SYSTEM ETFA2023
  (* Version 1.0, 2023-03-17, AK125171 *)
  APPLICATION ETFA2023App
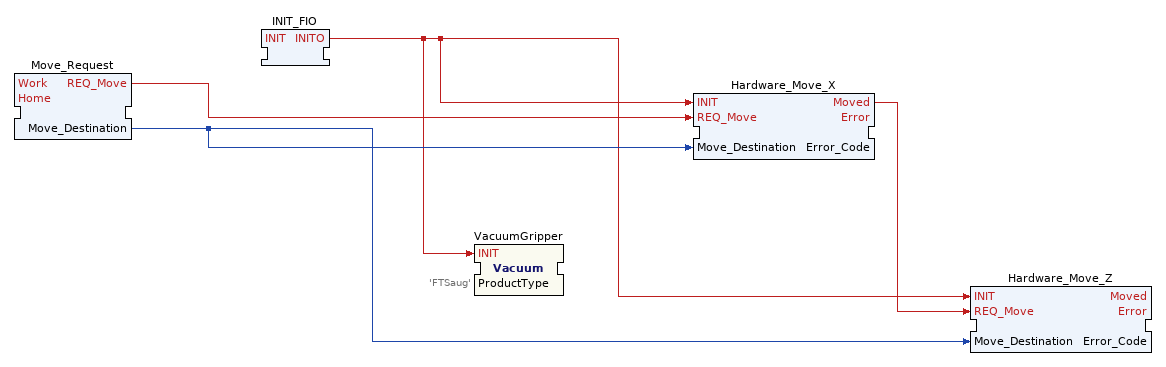
    FBS
      VacuumGripper : Vacuum(ProductType := 'FTSaug');
    END_FBS
    SUBAPPLICATION INIT_FIO
      EVENT_INPUT
        INIT;
      END_EVENT
      EVENT_OUTPUT
        INITO;
      END_EVENT
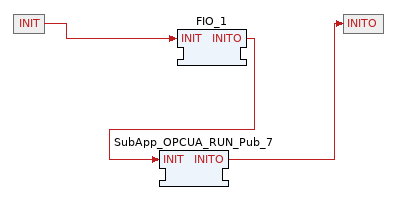
      SUBAPPLICATION SubApp_OPCUA_RUN_Pub_7
        EVENT_INPUT
          INIT;
        END_EVENT
        EVENT_OUTPUT
          INITO;
        END_EVENT
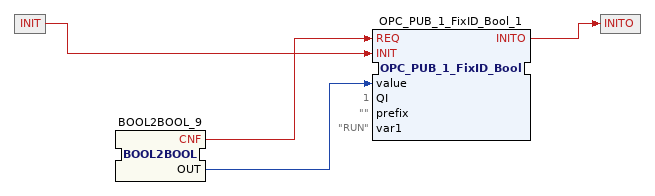
        FBS
          BOOL2BOOL_9 : BOOL2BOOL;
        END_FBS
        SUBAPPS
          OPC_PUB_1_FixID_Bool_1 : OPC_PUB_1_FixID_Bool(QI := 1, prefix := "", var1 := "RUN");
        END_SUBAPPS
        EVENT_CONNECTIONS
          BOOL2BOOL_9.CNF TO OPC_PUB_1_FixID_Bool_1.REQ;
          INIT TO OPC_PUB_1_FixID_Bool_1.INIT;
          OPC_PUB_1_FixID_Bool_1.INITO TO INITO;
        END_CONNECTIONS
        DATA_CONNECTIONS
          BOOL2BOOL_9.OUT TO OPC_PUB_1_FixID_Bool_1.value;
        END_CONNECTIONS
      END_SUBAPPLICATION
      SUBAPPLICATION FIO_1
        EVENT_INPUT
          INIT;
        END_EVENT
        EVENT_OUTPUT
          INITO;
        END_EVENT
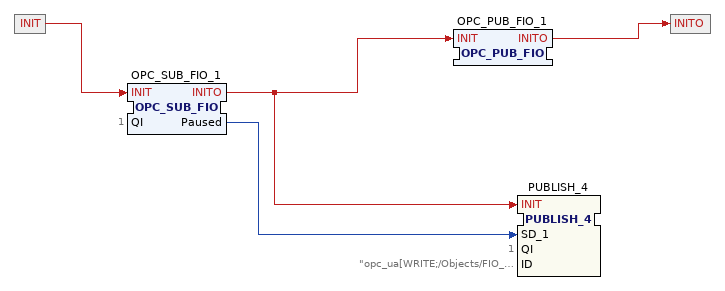
        FBS
          PUBLISH_4 : PUBLISH_4(QI := 1, ID := "opc_ua[WRITE;/Objects/FIO_Q_CameraPosition, 1:s=FIO_Q_CameraPosition;/Objects/FIO_Q_Pause, 1:s=FIO_Q_Pause;/Objects/FIO_Q_Reset, 1:s=FIO_Q_Reset;/Objects/FIO_Q_Run, 1:s=FIO_Q_Run]");
        END_FBS
        SUBAPPS
          OPC_PUB_FIO_1 : OPC_PUB_FIO;
          OPC_SUB_FIO_1 : OPC_SUB_FIO(QI := 1);
        END_SUBAPPS
        EVENT_CONNECTIONS
          OPC_SUB_FIO_1.INITO TO PUBLISH_4.INIT;
          OPC_SUB_FIO_1.INITO TO OPC_PUB_FIO_1.INIT;
          OPC_PUB_FIO_1.INITO TO INITO;
          INIT TO OPC_SUB_FIO_1.INIT;
        END_CONNECTIONS
        DATA_CONNECTIONS
          OPC_SUB_FIO_1.Paused TO PUBLISH_4.SD_1;
        END_CONNECTIONS
      END_SUBAPPLICATION
      EVENT_CONNECTIONS
        FIO_1.INITO TO SubApp_OPCUA_RUN_Pub_7.INIT;
        INIT TO FIO_1.INIT;
        SubApp_OPCUA_RUN_Pub_7.INITO TO INITO;
      END_CONNECTIONS
    END_SUBAPPLICATION
    SUBAPPLICATION Move_Request
      EVENT_INPUT
        Work;
        Home;
      END_EVENT
      EVENT_OUTPUT
        REQ_Move;
      END_EVENT
      VAR_OUTPUT
        Move_Destination : STRING;
      END_VAR
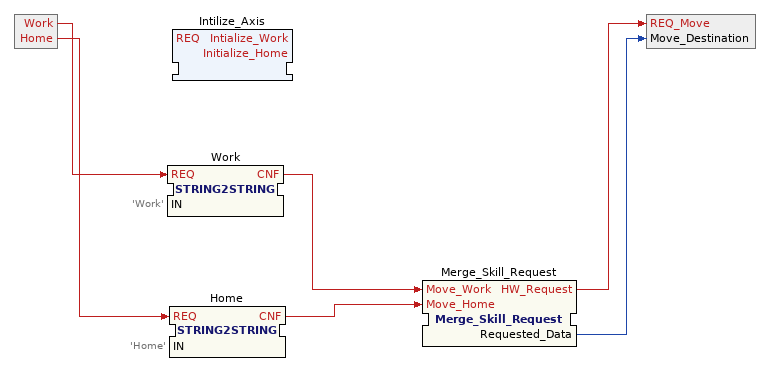
      FBS
        Work : STRING2STRING(IN := 'Work');
        Home : STRING2STRING(IN := 'Home');
        Merge_Skill_Request : Merge_Skill_Request;
      END_FBS
      SUBAPPLICATION Intilize_Axis
        EVENT_INPUT
          REQ;
        END_EVENT
        EVENT_OUTPUT
          Intialize_Work; (* Connect to Move_Work to intialize Work as start position else Connect to Move_Home to intialize Home as start position *)
          Initialize_Home;
        END_EVENT
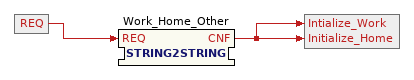
        FBS
          Work_Home_Other : STRING2STRING; (* Connect to Move_Work or Move_Home interface  of Instace Merge_Skill_Request *)
        END_FBS
        EVENT_CONNECTIONS
          REQ TO Work_Home_Other.REQ;
          Work_Home_Other.CNF TO Intialize_Work;
          Work_Home_Other.CNF TO Initialize_Home;
        END_CONNECTIONS
      END_SUBAPPLICATION
      EVENT_CONNECTIONS
        Work TO Work.REQ;
        Home TO Home.REQ;
        Work.CNF TO Merge_Skill_Request.Move_Work;
        Home.CNF TO Merge_Skill_Request.Move_Home;
        Merge_Skill_Request.HW_Request TO REQ_Move;
      END_CONNECTIONS
      DATA_CONNECTIONS
        Merge_Skill_Request.Requested_Data TO Move_Destination;
      END_CONNECTIONS
    END_SUBAPPLICATION
    SUBAPPLICATION Hardware_Move_X (* Hardware *)
      EVENT_INPUT
        INIT;
        REQ_Move;
      END_EVENT
      EVENT_OUTPUT
        Moved;
        Error;
      END_EVENT
      VAR_INPUT
        Move_Destination : STRING;
      END_VAR
      VAR_OUTPUT
        Error_Code : INT;
      END_VAR
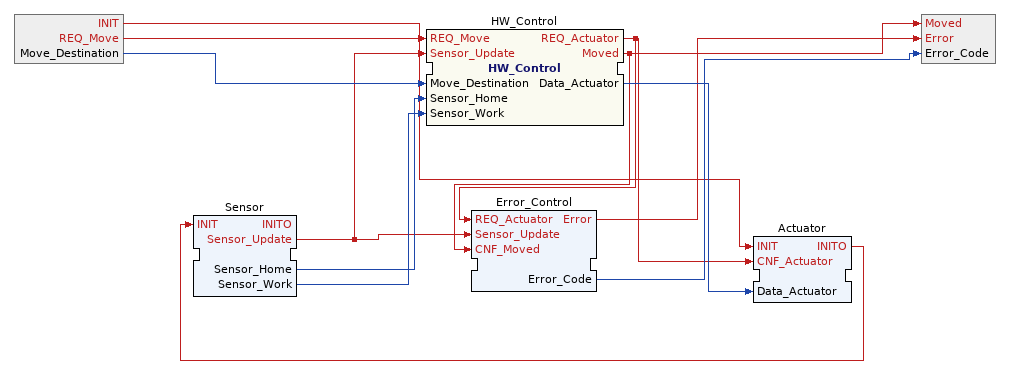
      FBS
        HW_Control : HW_Control;
      END_FBS
      SUBAPPLICATION Actuator
        EVENT_INPUT
          INIT;
          CNF_Actuator;
        END_EVENT
        EVENT_OUTPUT
          INITO;
        END_EVENT
        VAR_INPUT
          Data_Actuator : BOOL;
        END_VAR
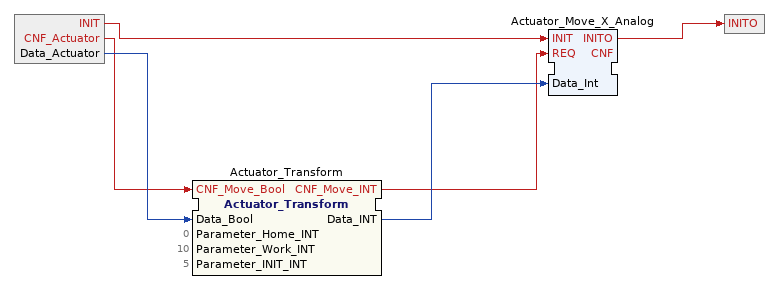
        FBS
          Actuator_Transform : Actuator_Transform(Parameter_Home_INT := 0, Parameter_Work_INT := 10, Parameter_INIT_INT := 5);
        END_FBS
        SUBAPPLICATION Actuator_Move_X_Analog
          EVENT_INPUT
            INIT;
            REQ;
          END_EVENT
          EVENT_OUTPUT
            INITO;
            CNF;
          END_EVENT
          VAR_INPUT
            Data_Int : INT;
          END_VAR
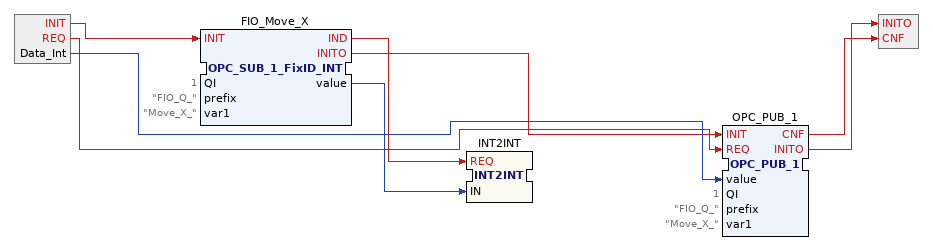
          FBS
            INT2INT : INT2INT;
          END_FBS
          SUBAPPS
            FIO_Move_X : OPC_SUB_1_FixID_INT(QI := 1, prefix := "FIO_Q_", var1 := "Move_X_");
            OPC_PUB_1 : OPC_PUB_1(QI := 1, prefix := "FIO_Q_", var1 := "Move_X_");
          END_SUBAPPS
          EVENT_CONNECTIONS
            INIT TO FIO_Move_X.INIT;
            FIO_Move_X.IND TO INT2INT.REQ;
            FIO_Move_X.INITO TO OPC_PUB_1.INIT;
            OPC_PUB_1.CNF TO CNF;
            OPC_PUB_1.INITO TO INITO;
            REQ TO OPC_PUB_1.REQ;
          END_CONNECTIONS
          DATA_CONNECTIONS
            Data_Int TO OPC_PUB_1.value;
            FIO_Move_X.value TO INT2INT.IN;
          END_CONNECTIONS
        END_SUBAPPLICATION
        EVENT_CONNECTIONS
          INIT TO Actuator_Move_X_Analog.INIT;
          Actuator_Move_X_Analog.INITO TO INITO;
          CNF_Actuator TO Actuator_Transform.CNF_Move_Bool;
          Actuator_Transform.CNF_Move_INT TO Actuator_Move_X_Analog.REQ;
        END_CONNECTIONS
        DATA_CONNECTIONS
          Data_Actuator TO Actuator_Transform.Data_Bool;
          Actuator_Transform.Data_INT TO Actuator_Move_X_Analog.Data_Int;
        END_CONNECTIONS
      END_SUBAPPLICATION
      SUBAPPLICATION Error_Control
        EVENT_INPUT
          REQ_Actuator;
          Sensor_Update;
          CNF_Moved;
        END_EVENT
        EVENT_OUTPUT
          Error;
        END_EVENT
        VAR_OUTPUT
          Error_Code : INT; (* Error_Code_1_For_Movement_Not_Started_Error_Code_2_For_Movement_Timing *)
        END_VAR
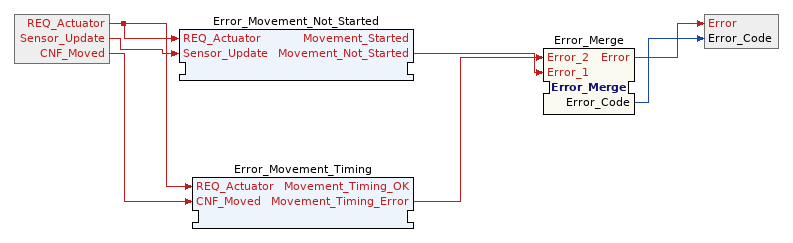
        FBS
          Error_Merge : Error_Merge;
        END_FBS
        SUBAPPLICATION Error_Movement_Not_Started
          EVENT_INPUT
            REQ_Actuator;
            Sensor_Update;
          END_EVENT
          EVENT_OUTPUT
            Movement_Started;
            Movement_Not_Started;
          END_EVENT
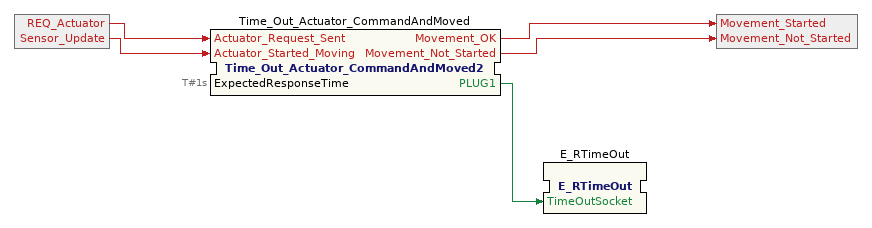
          FBS
            E_RTimeOut : E_RTimeOut;
            Time_Out_Actuator_CommandAndMoved : Time_Out_Actuator_CommandAndMoved2(ExpectedResponseTime := T#1s);
          END_FBS
          EVENT_CONNECTIONS
            REQ_Actuator TO Time_Out_Actuator_CommandAndMoved.Actuator_Request_Sent;
            Sensor_Update TO Time_Out_Actuator_CommandAndMoved.Actuator_Started_Moving;
            Time_Out_Actuator_CommandAndMoved.Movement_OK TO Movement_Started;
            Time_Out_Actuator_CommandAndMoved.Movement_Not_Started TO Movement_Not_Started;
          END_CONNECTIONS
          ADAPTER_CONNECTIONS
            Time_Out_Actuator_CommandAndMoved.PLUG1 TO E_RTimeOut.TimeOutSocket;
          END_CONNECTIONS
        END_SUBAPPLICATION
        SUBAPPLICATION Error_Movement_Timing
          EVENT_INPUT
            REQ_Actuator;
            CNF_Moved;
          END_EVENT
          EVENT_OUTPUT
            Movement_Timing_OK;
            Movement_Timing_Error;
          END_EVENT
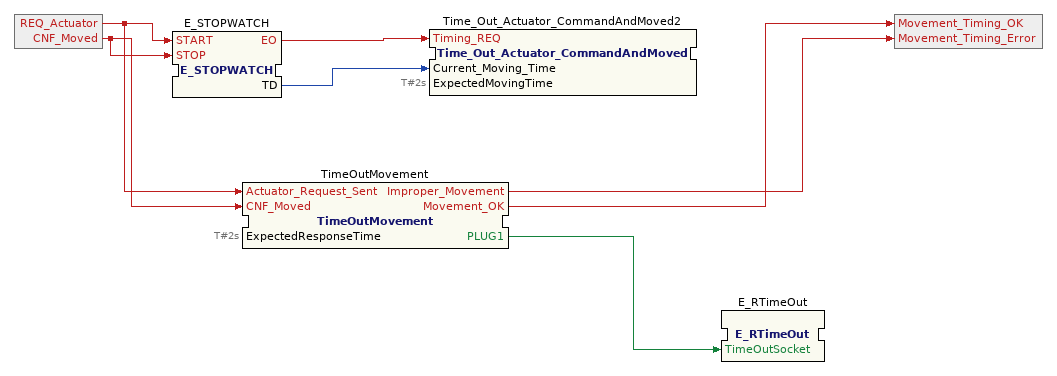
          FBS
            E_STOPWATCH : E_STOPWATCH;
            Time_Out_Actuator_CommandAndMoved2 : Time_Out_Actuator_CommandAndMoved(ExpectedMovingTime := T#2s);
            E_RTimeOut : E_RTimeOut;
            TimeOutMovement : TimeOutMovement(ExpectedResponseTime := T#2s);
          END_FBS
          EVENT_CONNECTIONS
            E_STOPWATCH.EO TO Time_Out_Actuator_CommandAndMoved2.Timing_REQ;
            REQ_Actuator TO TimeOutMovement.Actuator_Request_Sent;
            CNF_Moved TO TimeOutMovement.CNF_Moved;
            TimeOutMovement.Improper_Movement TO Movement_Timing_Error;
            TimeOutMovement.Movement_OK TO Movement_Timing_OK;
            REQ_Actuator TO E_STOPWATCH.START;
            CNF_Moved TO E_STOPWATCH.STOP;
          END_CONNECTIONS
          DATA_CONNECTIONS
            E_STOPWATCH.TD TO Time_Out_Actuator_CommandAndMoved2.Current_Moving_Time;
          END_CONNECTIONS
          ADAPTER_CONNECTIONS
            TimeOutMovement.PLUG1 TO E_RTimeOut.TimeOutSocket;
          END_CONNECTIONS
        END_SUBAPPLICATION
        EVENT_CONNECTIONS
          REQ_Actuator TO Error_Movement_Not_Started.REQ_Actuator;
          Sensor_Update TO Error_Movement_Not_Started.Sensor_Update;
          CNF_Moved TO Error_Movement_Timing.CNF_Moved;
          Error_Movement_Timing.Movement_Timing_Error TO Error_Merge.Error_2;
          Error_Merge.Error TO Error;
          Error_Movement_Not_Started.Movement_Not_Started TO Error_Merge.Error_1;
          REQ_Actuator TO Error_Movement_Timing.REQ_Actuator;
        END_CONNECTIONS
        DATA_CONNECTIONS
          Error_Merge.Error_Code TO Error_Code;
        END_CONNECTIONS
      END_SUBAPPLICATION
      SUBAPPLICATION Sensor
        EVENT_INPUT
          INIT;
        END_EVENT
        EVENT_OUTPUT
          INITO;
          Sensor_Update;
        END_EVENT
        VAR_OUTPUT
          Sensor_Home : BOOL;
          Sensor_Work : BOOL;
        END_VAR
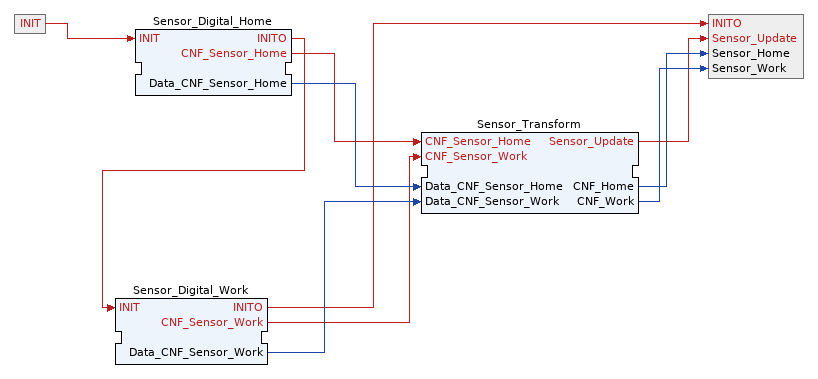
        SUBAPPLICATION Sensor_Digital_Work
          EVENT_INPUT
            INIT;
          END_EVENT
          EVENT_OUTPUT
            INITO;
            CNF_Sensor_Work;
          END_EVENT
          VAR_OUTPUT
            Data_CNF_Sensor_Work : BOOL;
          END_VAR
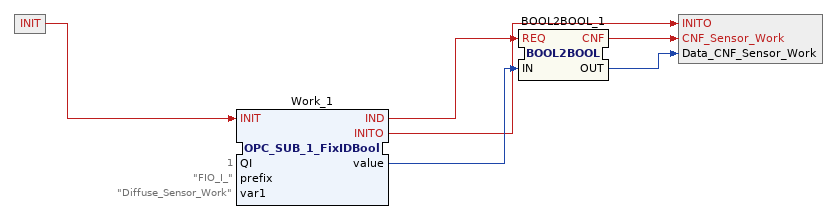
          FBS
            BOOL2BOOL_1 : BOOL2BOOL;
          END_FBS
          SUBAPPS
            Work_1 : OPC_SUB_1_FixIDBool(QI := 1, prefix := "FIO_I_", var1 := "Diffuse_Sensor_Work");
          END_SUBAPPS
          EVENT_CONNECTIONS
            Work_1.IND TO BOOL2BOOL_1.REQ;
            INIT TO Work_1.INIT;
            Work_1.INITO TO INITO;
            BOOL2BOOL_1.CNF TO CNF_Sensor_Work;
          END_CONNECTIONS
          DATA_CONNECTIONS
            Work_1.value TO BOOL2BOOL_1.IN;
            BOOL2BOOL_1.OUT TO Data_CNF_Sensor_Work;
          END_CONNECTIONS
        END_SUBAPPLICATION
        SUBAPPLICATION Sensor_Digital_Home
          EVENT_INPUT
            INIT;
          END_EVENT
          EVENT_OUTPUT
            INITO;
            CNF_Sensor_Home;
          END_EVENT
          VAR_OUTPUT
            Data_CNF_Sensor_Home : BOOL;
          END_VAR
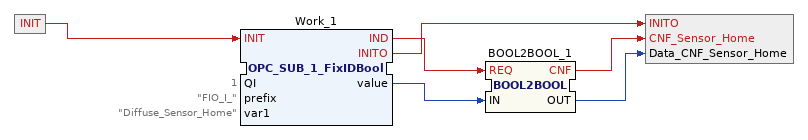
          FBS
            BOOL2BOOL_1 : BOOL2BOOL;
          END_FBS
          SUBAPPS
            Work_1 : OPC_SUB_1_FixIDBool(QI := 1, prefix := "FIO_I_", var1 := "Diffuse_Sensor_Home");
          END_SUBAPPS
          EVENT_CONNECTIONS
            Work_1.IND TO BOOL2BOOL_1.REQ;
            INIT TO Work_1.INIT;
            Work_1.INITO TO INITO;
            BOOL2BOOL_1.CNF TO CNF_Sensor_Home;
          END_CONNECTIONS
          DATA_CONNECTIONS
            Work_1.value TO BOOL2BOOL_1.IN;
            BOOL2BOOL_1.OUT TO Data_CNF_Sensor_Home;
          END_CONNECTIONS
        END_SUBAPPLICATION
        SUBAPPLICATION Sensor_Transform
          EVENT_INPUT
            CNF_Sensor_Home;
            CNF_Sensor_Work;
          END_EVENT
          EVENT_OUTPUT
            Sensor_Update;
          END_EVENT
          VAR_INPUT
            Data_CNF_Sensor_Home : BOOL;
            Data_CNF_Sensor_Work : BOOL;
          END_VAR
          VAR_OUTPUT
            CNF_Home : BOOL;
            CNF_Work : BOOL;
          END_VAR
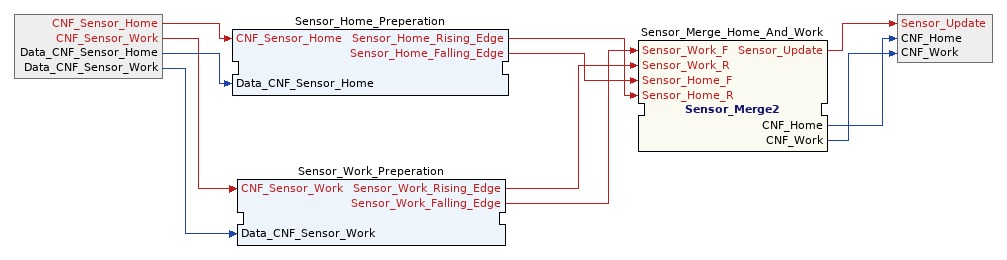
          FBS
            Sensor_Merge_Home_And_Work : Sensor_Merge2;
          END_FBS
          SUBAPPLICATION Sensor_Work_Preperation
            EVENT_INPUT
              CNF_Sensor_Work;
            END_EVENT
            EVENT_OUTPUT
              Sensor_Work_Rising_Edge;
              Sensor_Work_Falling_Edge;
            END_EVENT
            VAR_INPUT
              Data_CNF_Sensor_Work : BOOL;
            END_VAR
            FBS
              E_F_TRIG_Work : E_F_TRIG;
              E_R_TRIG_Work : E_R_TRIG;
            END_FBS
            EVENT_CONNECTIONS
              E_F_TRIG_Work.EO TO Sensor_Work_Falling_Edge;
              E_R_TRIG_Work.EO TO Sensor_Work_Rising_Edge;
              CNF_Sensor_Work TO E_R_TRIG_Work.EI;
              CNF_Sensor_Work TO E_F_TRIG_Work.EI;
            END_CONNECTIONS
            DATA_CONNECTIONS
              Data_CNF_Sensor_Work TO E_R_TRIG_Work.QI;
              Data_CNF_Sensor_Work TO E_F_TRIG_Work.QI;
            END_CONNECTIONS
          END_SUBAPPLICATION
          SUBAPPLICATION Sensor_Home_Preperation
            EVENT_INPUT
              CNF_Sensor_Home;
            END_EVENT
            EVENT_OUTPUT
              Sensor_Home_Rising_Edge;
              Sensor_Home_Falling_Edge;
            END_EVENT
            VAR_INPUT
              Data_CNF_Sensor_Home : BOOL;
            END_VAR
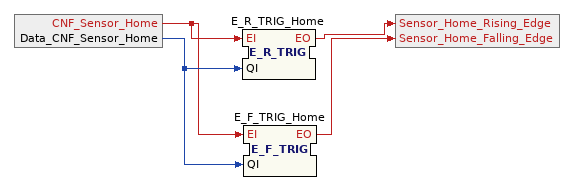
            FBS
              E_F_TRIG_Home : E_F_TRIG;
              E_R_TRIG_Home : E_R_TRIG;
            END_FBS
            EVENT_CONNECTIONS
              E_F_TRIG_Home.EO TO Sensor_Home_Falling_Edge;
              E_R_TRIG_Home.EO TO Sensor_Home_Rising_Edge;
              CNF_Sensor_Home TO E_R_TRIG_Home.EI;
              CNF_Sensor_Home TO E_F_TRIG_Home.EI;
            END_CONNECTIONS
            DATA_CONNECTIONS
              Data_CNF_Sensor_Home TO E_R_TRIG_Home.QI;
              Data_CNF_Sensor_Home TO E_F_TRIG_Home.QI;
            END_CONNECTIONS
          END_SUBAPPLICATION
          EVENT_CONNECTIONS
            Sensor_Merge_Home_And_Work.Sensor_Update TO Sensor_Update;
            Sensor_Work_Preperation.Sensor_Work_Falling_Edge TO Sensor_Merge_Home_And_Work.Sensor_Work_F;
            Sensor_Work_Preperation.Sensor_Work_Rising_Edge TO Sensor_Merge_Home_And_Work.Sensor_Work_R;
            CNF_Sensor_Work TO Sensor_Work_Preperation.CNF_Sensor_Work;
            Sensor_Home_Preperation.Sensor_Home_Falling_Edge TO Sensor_Merge_Home_And_Work.Sensor_Home_F;
            Sensor_Home_Preperation.Sensor_Home_Rising_Edge TO Sensor_Merge_Home_And_Work.Sensor_Home_R;
            CNF_Sensor_Home TO Sensor_Home_Preperation.CNF_Sensor_Home;
          END_CONNECTIONS
          DATA_CONNECTIONS
            Sensor_Merge_Home_And_Work.CNF_Home TO CNF_Home;
            Sensor_Merge_Home_And_Work.CNF_Work TO CNF_Work;
            Data_CNF_Sensor_Work TO Sensor_Work_Preperation.Data_CNF_Sensor_Work;
            Data_CNF_Sensor_Home TO Sensor_Home_Preperation.Data_CNF_Sensor_Home;
          END_CONNECTIONS
        END_SUBAPPLICATION
        EVENT_CONNECTIONS
          Sensor_Digital_Home.INITO TO Sensor_Digital_Work.INIT;
          INIT TO Sensor_Digital_Home.INIT;
          Sensor_Digital_Work.INITO TO INITO;
          Sensor_Digital_Work.CNF_Sensor_Work TO Sensor_Transform.CNF_Sensor_Work;
          Sensor_Digital_Home.CNF_Sensor_Home TO Sensor_Transform.CNF_Sensor_Home;
          Sensor_Transform.Sensor_Update TO Sensor_Update;
        END_CONNECTIONS
        DATA_CONNECTIONS
          Sensor_Digital_Work.Data_CNF_Sensor_Work TO Sensor_Transform.Data_CNF_Sensor_Work;
          Sensor_Digital_Home.Data_CNF_Sensor_Home TO Sensor_Transform.Data_CNF_Sensor_Home;
          Sensor_Transform.CNF_Work TO Sensor_Work;
          Sensor_Transform.CNF_Home TO Sensor_Home;
        END_CONNECTIONS
      END_SUBAPPLICATION
      EVENT_CONNECTIONS
        HW_Control.REQ_Actuator TO Actuator.CNF_Actuator;
        HW_Control.REQ_Actuator TO Error_Control.REQ_Actuator;
        HW_Control.Moved TO Error_Control.CNF_Moved;
        REQ_Move TO HW_Control.REQ_Move;
        HW_Control.Moved TO Moved;
        Error_Control.Error TO Error;
        INIT TO Actuator.INIT;
        Actuator.INITO TO Sensor.INIT;
        Sensor.Sensor_Update TO Error_Control.Sensor_Update;
        Sensor.Sensor_Update TO HW_Control.Sensor_Update;
      END_CONNECTIONS
      DATA_CONNECTIONS
        HW_Control.Data_Actuator TO Actuator.Data_Actuator;
        Move_Destination TO HW_Control.Move_Destination;
        Error_Control.Error_Code TO Error_Code;
        Sensor.Sensor_Home TO HW_Control.Sensor_Home;
        Sensor.Sensor_Work TO HW_Control.Sensor_Work;
      END_CONNECTIONS
    END_SUBAPPLICATION
    SUBAPPLICATION Hardware_Move_Z (* Hardware *)
      EVENT_INPUT
        INIT;
        REQ_Move;
      END_EVENT
      EVENT_OUTPUT
        Moved;
        Error;
      END_EVENT
      VAR_INPUT
        Move_Destination : STRING;
      END_VAR
      VAR_OUTPUT
        Error_Code : INT;
      END_VAR
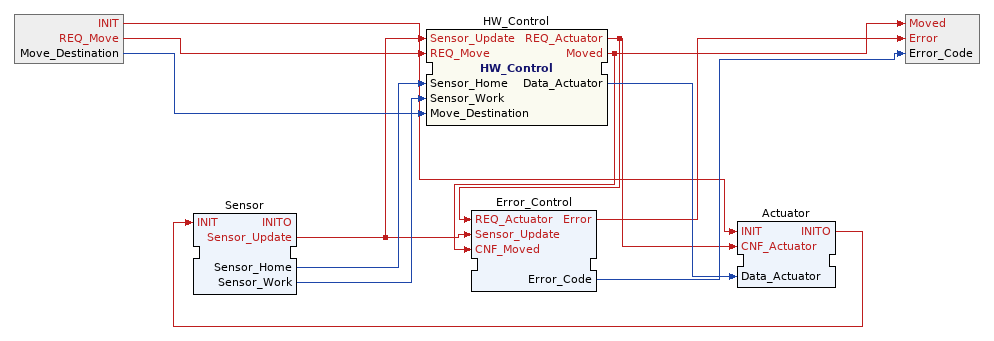
      FBS
        HW_Control : HW_Control;
      END_FBS
      SUBAPPLICATION Actuator
        EVENT_INPUT
          INIT;
          CNF_Actuator;
        END_EVENT
        EVENT_OUTPUT
          INITO;
        END_EVENT
        VAR_INPUT
          Data_Actuator : BOOL;
        END_VAR
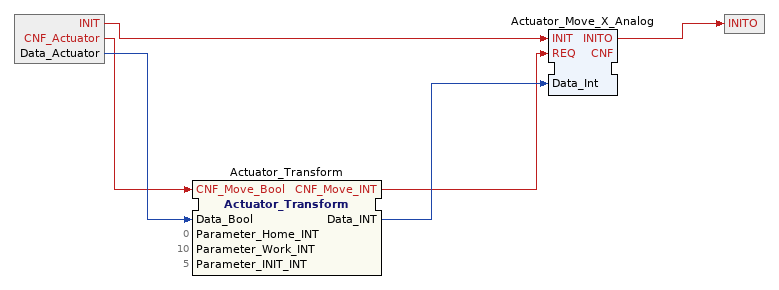
        FBS
          Actuator_Transform : Actuator_Transform(Parameter_Home_INT := 0, Parameter_Work_INT := 10, Parameter_INIT_INT := 5);
        END_FBS
        SUBAPPLICATION Actuator_Move_X_Analog
          EVENT_INPUT
            INIT;
            REQ;
          END_EVENT
          EVENT_OUTPUT
            INITO;
            CNF;
          END_EVENT
          VAR_INPUT
            Data_Int : INT;
          END_VAR
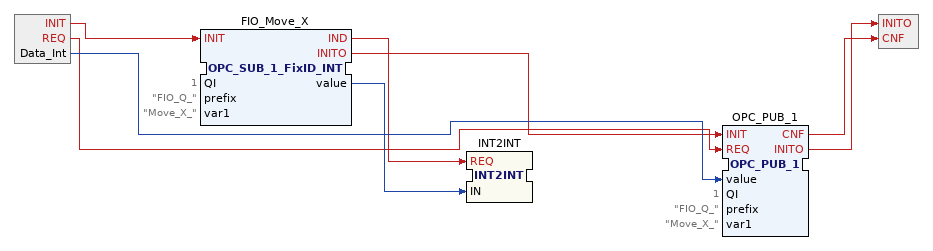
          FBS
            INT2INT : INT2INT;
          END_FBS
          SUBAPPS
            FIO_Move_X : OPC_SUB_1_FixID_INT(QI := 1, prefix := "FIO_Q_", var1 := "Move_X_");
            OPC_PUB_1 : OPC_PUB_1(QI := 1, prefix := "FIO_Q_", var1 := "Move_X_");
          END_SUBAPPS
          EVENT_CONNECTIONS
            INIT TO FIO_Move_X.INIT;
            FIO_Move_X.IND TO INT2INT.REQ;
            FIO_Move_X.INITO TO OPC_PUB_1.INIT;
            OPC_PUB_1.CNF TO CNF;
            OPC_PUB_1.INITO TO INITO;
            REQ TO OPC_PUB_1.REQ;
          END_CONNECTIONS
          DATA_CONNECTIONS
            Data_Int TO OPC_PUB_1.value;
            FIO_Move_X.value TO INT2INT.IN;
          END_CONNECTIONS
        END_SUBAPPLICATION
        EVENT_CONNECTIONS
          INIT TO Actuator_Move_X_Analog.INIT;
          Actuator_Move_X_Analog.INITO TO INITO;
          CNF_Actuator TO Actuator_Transform.CNF_Move_Bool;
          Actuator_Transform.CNF_Move_INT TO Actuator_Move_X_Analog.REQ;
        END_CONNECTIONS
        DATA_CONNECTIONS
          Data_Actuator TO Actuator_Transform.Data_Bool;
          Actuator_Transform.Data_INT TO Actuator_Move_X_Analog.Data_Int;
        END_CONNECTIONS
      END_SUBAPPLICATION
      SUBAPPLICATION Error_Control
        EVENT_INPUT
          REQ_Actuator;
          Sensor_Update;
          CNF_Moved;
        END_EVENT
        EVENT_OUTPUT
          Error;
        END_EVENT
        VAR_OUTPUT
          Error_Code : INT; (* Error_Code_1_For_Movement_Not_Started_Error_Code_2_For_Movement_Timing *)
        END_VAR
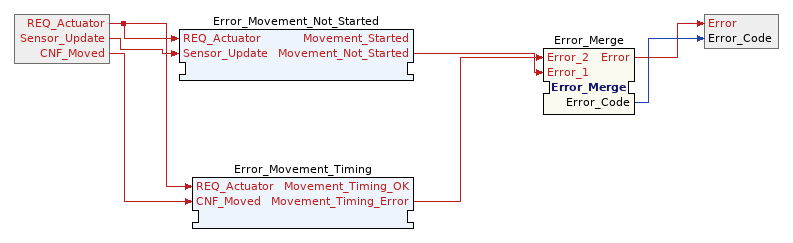
        FBS
          Error_Merge : Error_Merge;
        END_FBS
        SUBAPPLICATION Error_Movement_Not_Started
          EVENT_INPUT
            REQ_Actuator;
            Sensor_Update;
          END_EVENT
          EVENT_OUTPUT
            Movement_Started;
            Movement_Not_Started;
          END_EVENT
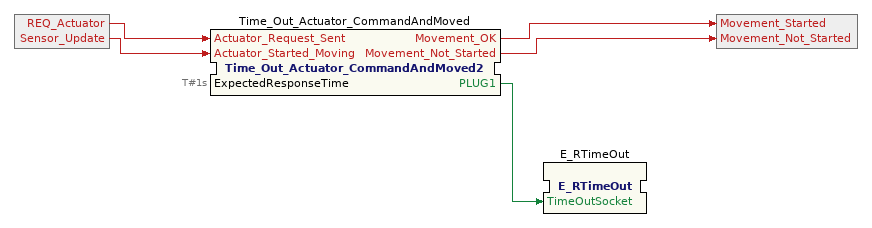
          FBS
            E_RTimeOut : E_RTimeOut;
            Time_Out_Actuator_CommandAndMoved : Time_Out_Actuator_CommandAndMoved2(ExpectedResponseTime := T#1s);
          END_FBS
          EVENT_CONNECTIONS
            REQ_Actuator TO Time_Out_Actuator_CommandAndMoved.Actuator_Request_Sent;
            Sensor_Update TO Time_Out_Actuator_CommandAndMoved.Actuator_Started_Moving;
            Time_Out_Actuator_CommandAndMoved.Movement_OK TO Movement_Started;
            Time_Out_Actuator_CommandAndMoved.Movement_Not_Started TO Movement_Not_Started;
          END_CONNECTIONS
          ADAPTER_CONNECTIONS
            Time_Out_Actuator_CommandAndMoved.PLUG1 TO E_RTimeOut.TimeOutSocket;
          END_CONNECTIONS
        END_SUBAPPLICATION
        SUBAPPLICATION Error_Movement_Timing
          EVENT_INPUT
            REQ_Actuator;
            CNF_Moved;
          END_EVENT
          EVENT_OUTPUT
            Movement_Timing_OK;
            Movement_Timing_Error;
          END_EVENT
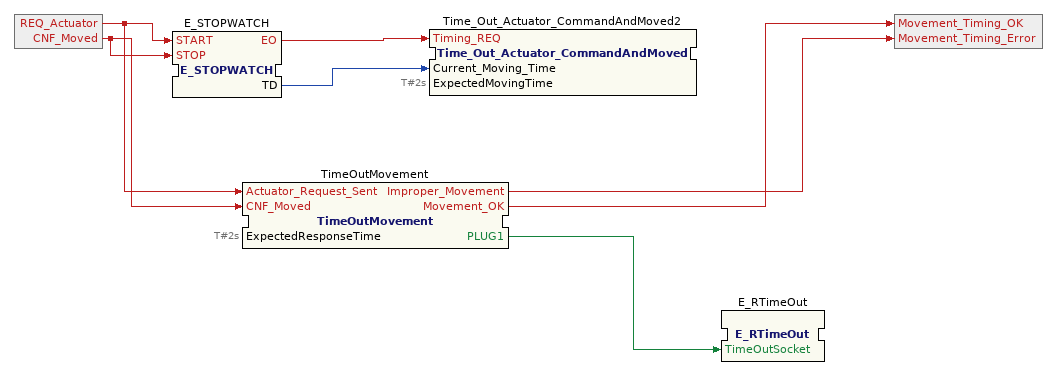
          FBS
            E_STOPWATCH : E_STOPWATCH;
            Time_Out_Actuator_CommandAndMoved2 : Time_Out_Actuator_CommandAndMoved(ExpectedMovingTime := T#2s);
            E_RTimeOut : E_RTimeOut;
            TimeOutMovement : TimeOutMovement(ExpectedResponseTime := T#2s);
          END_FBS
          EVENT_CONNECTIONS
            E_STOPWATCH.EO TO Time_Out_Actuator_CommandAndMoved2.Timing_REQ;
            REQ_Actuator TO TimeOutMovement.Actuator_Request_Sent;
            CNF_Moved TO TimeOutMovement.CNF_Moved;
            TimeOutMovement.Improper_Movement TO Movement_Timing_Error;
            TimeOutMovement.Movement_OK TO Movement_Timing_OK;
            REQ_Actuator TO E_STOPWATCH.START;
            CNF_Moved TO E_STOPWATCH.STOP;
          END_CONNECTIONS
          DATA_CONNECTIONS
            E_STOPWATCH.TD TO Time_Out_Actuator_CommandAndMoved2.Current_Moving_Time;
          END_CONNECTIONS
          ADAPTER_CONNECTIONS
            TimeOutMovement.PLUG1 TO E_RTimeOut.TimeOutSocket;
          END_CONNECTIONS
        END_SUBAPPLICATION
        EVENT_CONNECTIONS
          REQ_Actuator TO Error_Movement_Not_Started.REQ_Actuator;
          Sensor_Update TO Error_Movement_Not_Started.Sensor_Update;
          CNF_Moved TO Error_Movement_Timing.CNF_Moved;
          Error_Movement_Timing.Movement_Timing_Error TO Error_Merge.Error_2;
          Error_Merge.Error TO Error;
          Error_Movement_Not_Started.Movement_Not_Started TO Error_Merge.Error_1;
          REQ_Actuator TO Error_Movement_Timing.REQ_Actuator;
        END_CONNECTIONS
        DATA_CONNECTIONS
          Error_Merge.Error_Code TO Error_Code;
        END_CONNECTIONS
      END_SUBAPPLICATION
      SUBAPPLICATION Sensor
        EVENT_INPUT
          INIT;
        END_EVENT
        EVENT_OUTPUT
          INITO;
          Sensor_Update;
        END_EVENT
        VAR_OUTPUT
          Sensor_Home : BOOL;
          Sensor_Work : BOOL;
        END_VAR
